FUNCTION_BLOCK FB_PWT1System
VAR_INPUT
END_VAR
VAR_OUTPUT
END_VAR
VAR
END_VAR

END_FUNCTION_BLOCK

(* stored: Version 1.1.0.1, ProductVersion 3.1.4024.10
   POU FB_PWT1System: Id {61964d8e-51ba-4d03-8634-2a417c9ac9b4}, SpecialFunc None *)
